//{{V2}}
FUNCTION FC1
TITLE= <Title of FC>


AUTHOR:nb
FAMILY:nb
NAME:nb
VERSION:1.0


VAR_INPUT
END_VAR

VAR_OUTPUT
END_VAR

VAR_IN_OUT
END_VAR

VAR_TEMP
END_VAR
BEGIN

NETWORK
TITLE=
//{{k}}

       A    I         0.0
       =    Q         0.1

END_FUNCTION
